// TIA Portal V20 export
FUNCTION "FC_OUTPUT_MAP" : Void   // FC102, LAD
{ S7_Optimized_Access := 'TRUE' }
// stored: AutoNumber false, SetENOAutomatically false
   VAR_TEMP
      LOOP : Int;
      Value : Byte;
   END_VAR
BEGIN

REGION Network 1 (SCL): OUTPUT900BYTE
   FOR #LOOP := 0 TO 900 BY 1 DO
       #Value := PEEK(area := 16#84, dbNumber := 16, byteOffset := #LOOP);
       POKE(area:=16#82,dbNumber:=0, byteOffset:=#LOOP,value:=#Value);
   END_FOR;
END_REGION
END_FUNCTION
